(* IEC 61131-3 sources: com.logicals.lc3.webinar/usRTS_RPMControl_iSOC/src_FB_LIB_SAFE/Numeric/INT, 8 files *)

(* ---- wADD_INT_2.iecst ---- *)
NAMESPACE logicals.web.standard
NAMESPACE numeric

/*
 * Function block wrapper for IEC 61131-3 ADD<br>
 * IN1 =  1st value (INT)<br>
 * IN2 =  2nd value (INT)<br>
 * OUT = Sum of all input values (INT)<br>
 */
FUNCTION_BLOCK wADD_INT_2
	{ vNameAlignment:="center"; altName:="+"; bgColor:="LightPink"; width:=40; hideIONames; }
	VAR_INPUT
		IN1 : INT;
		IN2 : INT;
	END_VAR
	VAR_OUTPUT
		OUT : INT;
	END_VAR

	OUT := ADD(IN1:=IN1, IN2:=IN2, ENO=>ENO);
END_FUNCTION_BLOCK

END_NAMESPACE
END_NAMESPACE

(* ---- wADD_INT_3.iecst ---- *)
NAMESPACE logicals.web.standard
NAMESPACE numeric

/*
 * Function block wrapper for IEC 61131-3 ADD<br>
 * IN1 =  1st value (INT)<br>
 * IN2 =  2nd value (INT)<br>
 * IN3 =  3rd value (INT)<br>
 * OUT = Sum of all input values (INT)<br>
 */
FUNCTION_BLOCK wADD_INT_3
	{ vNameAlignment:="center"; altName:="+"; bgColor:="LightPink"; width:=40; hideIONames; }
	VAR_INPUT
		IN1 : INT;
		IN2 : INT;
		IN3 : INT;
	END_VAR
	VAR_OUTPUT
		OUT : INT;
	END_VAR

	OUT := ADD(IN1:=IN1, IN2:=IN2, IN3:=IN3, ENO=>ENO);
END_FUNCTION_BLOCK

END_NAMESPACE
END_NAMESPACE

(* ---- wADD_INT_4.iecst ---- *)
NAMESPACE logicals.web.standard
NAMESPACE numeric

/*
 * Function block wrapper for IEC 61131-3 ADD<br>
 * IN1 =  1st value (INT)<br>
 * IN2 =  2nd value (INT)<br>
 * IN3 =  3rd value (INT)<br>
 * IN4 =  4th value (INT)<br>
 * OUT = Sum of all input values (INT)<br>
 */
FUNCTION_BLOCK wADD_INT_4
	{ vNameAlignment:="center"; altName:="+"; bgColor:="LightPink"; width:=40; hideIONames; }
	VAR_INPUT
		IN1 : INT;
		IN2 : INT;
		IN3 : INT;
		IN4 : INT;
	END_VAR
	VAR_OUTPUT
		OUT : INT;
	END_VAR

	OUT := ADD(IN1:=IN1, IN2:=IN2, IN3:=IN3, IN4:=IN4, ENO=>ENO);
END_FUNCTION_BLOCK

END_NAMESPACE
END_NAMESPACE

(* ---- wDIV_INT.iecst ---- *)
NAMESPACE logicals.web.standard
NAMESPACE numeric

/*
 * Function block wrapper for IEC 61131-3 DIV<br>
 * IN1 =  1st value (INT)<br>
 * IN2 =  2nd value (INT)<br>
 * OUT = quotient of IN1 divided by IN2 (INT)<br>
 */
FUNCTION_BLOCK wDIV_INT
	{ vNameAlignment:="center"; altName:="/"; bgColor:="LightPink"; width:=40; hideIONames; }
	VAR_INPUT
		IN1 : INT;
		IN2 : INT;
	END_VAR
	VAR_OUTPUT
		OUT : INT;
	END_VAR

	OUT := DIV(IN1:=IN1, IN2:=IN2, ENO=>ENO);
END_FUNCTION_BLOCK

END_NAMESPACE
END_NAMESPACE

(* ---- wMUL_INT_2.iecst ---- *)
NAMESPACE logicals.web.standard
NAMESPACE numeric

/*
 * Function block wrapper for IEC 61131-3 MUL<br>
 * IN1 =  1st value (INT)<br>
 * IN2 =  2nd value (INT)<br>
 * OUT = Product of multiplication of all inputs (INT)<br>
 */
FUNCTION_BLOCK wMUL_INT_2
	{ vNameAlignment:="center"; altName:="*"; bgColor:="LightPink"; width:=40; hideIONames; }
	VAR_INPUT
		IN1 : INT;
		IN2 : INT;
	END_VAR
	VAR_OUTPUT
		OUT : INT;
	END_VAR

	OUT := MUL(IN1:=IN1, IN2:=IN2, ENO=>ENO);
END_FUNCTION_BLOCK

END_NAMESPACE
END_NAMESPACE

(* ---- wMUL_INT_3.iecst ---- *)
NAMESPACE logicals.web.standard
NAMESPACE numeric

/*
 * Function block wrapper for IEC 61131-3 MUL<br>
 * IN1 =  1st value (INT)<br>
 * IN2 =  2nd value (INT)<br>
 * IN3 =  3rd value (INT)<br>
 * OUT = Product of multiplication of all inputs (INT)<br>
 */
FUNCTION_BLOCK wMUL_INT_3
	{ vNameAlignment:="center"; altName:="*"; bgColor:="LightPink"; width:=40; hideIONames; }
	VAR_INPUT
		IN1 : INT;
		IN2 : INT;
		IN3 : INT;
	END_VAR
	VAR_OUTPUT
		OUT : INT;
	END_VAR

	OUT := MUL(IN1:=IN1, IN2:=IN2, IN3:=IN3, ENO=>ENO);
END_FUNCTION_BLOCK

END_NAMESPACE
END_NAMESPACE

(* ---- wMUL_INT_4.iecst ---- *)
NAMESPACE logicals.web.standard
NAMESPACE numeric

/*
 * Function block wrapper for IEC 61131-3 MUL<br>
 * IN1 =  1st value (INT)<br>
 * IN2 =  2nd value (INT)<br>
 * IN3 =  3rd value (INT)<br>
 * IN4 =  4th value (INT)<br>
 * OUT = Product of multiplication of all inputs (INT)<br>
 */
FUNCTION_BLOCK wMUL_INT_4
	{ vNameAlignment:="center"; altName:="*"; bgColor:="LightPink"; width:=40; hideIONames; }
	VAR_INPUT
		IN1 : INT;
		IN2 : INT;
		IN3 : INT;
		IN4 : INT;
	END_VAR
	VAR_OUTPUT
		OUT : INT;
	END_VAR

	OUT := MUL(IN1:=IN1, IN2:=IN2, IN3:=IN3, IN4:=IN4, ENO=>ENO);
END_FUNCTION_BLOCK

END_NAMESPACE
END_NAMESPACE

(* ---- wSUB_INT.iecst ---- *)
NAMESPACE logicals.web.standard
NAMESPACE numeric

/*
 * Function block wrapper for IEC 61131-3 SUB<br>
 * IN1 =  1st value (INT)<br>
 * IN2 =  2nd value (INT)<br>
 * OUT = IN1 minus IN2 (INT)<br>
 */
FUNCTION_BLOCK wSUB_INT
	{ vNameAlignment:="center"; altName:="-"; bgColor:="LightPink"; width:=40; hideIONames; }
	VAR_INPUT
		IN1 : INT;
		IN2 : INT;
	END_VAR
	VAR_OUTPUT
		OUT : INT;
	END_VAR

	OUT := SUB(IN1:=IN1, IN2:=IN2, ENO=>ENO);
END_FUNCTION_BLOCK

END_NAMESPACE
END_NAMESPACE
